INTERFACE I_MutBinArg EXTENDS I_BinArg

PROPERTY Val : LWORD
SET
END_SET
END_PROPERTY

END_INTERFACE

(* stored: Version 1.1.0.1
   Itf I_MutBinArg: Id {7442cc50-5d45-4263-8234-371a76f710e8}
   Property Val: Id {e849d140-d716-49c4-a3e1-686d4fc39b81}
   Set Set: Id {b24aa621-5f63-4daf-9228-4e784aced44c} *)
